Fanuc KAREL source: IO0200.KL

PROGRAM IO0200
%NOLOCKGROUP
ROUTINE RTEST
VAR
L1 : ARRAY[3] OF INTEGER;L2 : XYZWPR
L3 : JOINTPOS9
L4 : POSITION
A:BOOLEAN
S1:INTEGER
B:REAL
C:BOOLEAN
D:REAL
BEGIN
--
--
A=TRUE
L1[1]=2
C=TRUE
D=1.0
SET_POS_REG(1,L2,S1,1)
END RTEST
BEGIN
RTEST
END IO0200
